PROGRAM confirmSetInicio
VAR
END_VAR

gvl.progInicio[gvl.actEst]:= 'DT#20';
gvl.progInicio[gvl.actEst]:= concat(gvl.progInicio[gvl.actEst],gvl.ano);
gvl.progInicio[gvl.actEst]:= concat(gvl.progInicio[gvl.actEst],'-');
gvl.progInicio[gvl.actEst]:= concat(gvl.progInicio[gvl.actEst],gvl.mes);
gvl.progInicio[gvl.actEst]:= concat(gvl.progInicio[gvl.actEst],'-');
gvl.progInicio[gvl.actEst]:= concat(gvl.progInicio[gvl.actEst],gvl.dia);
gvl.progInicio[gvl.actEst]:= concat(gvl.progInicio[gvl.actEst],'-');
gvl.progInicio[gvl.actEst]:= concat(gvl.progInicio[gvl.actEst],gvl.hora);
gvl.progInicio[gvl.actEst]:= concat(gvl.progInicio[gvl.actEst],':');
gvl.progInicio[gvl.actEst]:= concat(gvl.progInicio[gvl.actEst],gvl.minuto);
gvl.progInicio[gvl.actEst]:= concat(gvl.progInicio[gvl.actEst],':0');

END_PROGRAM

(* stored: Version 1.1.0.1, ProductVersion 3.1.4024.12
   POU confirmSetInicio: Id {798cbf82-934b-4c29-9928-68e4d06c4347}, SpecialFunc None *)
